(* CODESYS project WS11.project
   Title: WS11
   Version: 1.2.0
   Company: TTControl S.r.l.

Project tree, tasks and I/O mapping:
  Device : HY-TTC 580, TTControl, order no. n/a, version 1.8.0.0
    application Application
      libraries: Standard, * (System); Base Control Library Unsafe, 0.4.0.2 (TTControl); lib500_can2, 0.2.0.5 (TTControl); lib500, 1.8.0.0 (TTControl); lib500_types, 1.8.0.0 (TTControl); lib500_syscom, 1.8.0.0 (TTControl)
      task MainTask (cyclic, interval t#10ms, priority 2, watchdog t#10ms x 1) calls PLC_PRG
      task _ErrorCallback (externalevent, external event ErrorCallback, priority 1) calls _ErrorCB_PRG
      task _NotificationCallback (externalevent, external event NotificationCallback, priority 0) calls _NotificationCB_PRG
      program PLC_PRG [ST]
      program _ErrorCB_PRG [ST]
      program _NotificationCB_PRG [ST]
      global variables GVL
      program ReadMe [ST]
      program Disclaimer [ST]
      data type t_Power
      data type t_PWM
      global variables CONSTANTS
    CANs : CANs, TTControl, order no. n/a, version 1.8.0.0
      CAN0 : CAN0, TTControl, order no. n/a, version 1.8.0.0
      CAN1 : CAN1, TTControl, order no. n/a, version 1.8.0.0
          settings: Baudrate = 250
      CAN2 : CAN2, TTControl, order no. n/a, version 1.8.0.0
      CAN3 : CAN3, TTControl, order no. n/a, version 1.8.0.0
      CAN4 : CAN4, TTControl, order no. n/a, version 1.8.0.0
      CAN5 : CAN5, TTControl, order no. n/a, version 1.8.0.0
      CAN6 : CAN6, TTControl, order no. n/a, version 1.8.0.0
    System : System, TTControl, order no. n/a, version 1.8.0.0
        output Application.gPowerStage.Set.state : BYTE  // mode
        input  Application.gPowerStage.Set.error : WORD  // error
        output Application.gSafetySwitch0.Set.state : BYTE  // mode
        input  Application.gSafetySwitch0.Set.error : WORD  // error
        output Application.gSensorSupply.Set.state : BYTE  // mode
        input  Application.gSensorSupply.Set.error : WORD  // error
        input  Application.gDiagState : lib500_types.DIAG_STATUS  // diag_status
        input  Application.gSafetySwitch0.Feedback : lib500_types.IO_ADC_STATUS  // SSW0
        input  Application.gSensorSupply.Feedback : lib500_types.IO_ADC_STATUS  // SSUP0
        input  Application.gPowerStage.Get : lib500_types.IO_POWER_STATUS  // Powerstage
        input  Application.gSafetySwitch0.Get : lib500_types.IO_POWER_STATUS  // SSW0
        input  Application.gSensorSupply.Get : lib500_types.IO_POWER_STATUS  // SSUP0
        unmapped channels: mode, error, mode, error, mode, error, mode, error, shutdown, error, enable_error_group_0, enable_error_group_1, enable_error_group_2, safe_state, error, driver_init_error, UBAT, Terminal_15, WakeUp, Temperature, SSW1, SSW2, SSUP1, SSUP2, status, write, boot_error, trigger_error, SSW1, SSW2, SSUP1, SSUP2, Terminal_15, WakeUp, ExtShutOff0, ExtShutOff1, ExtShutOff2
      Analog_Inputs_2Mode_10V : AIN_2Mode_10V, TTControl, order no. n/a, version 1.8.0.0
        Pin 107
          PotRed : IoDrvADC2Mode10, TTControl, order no. n/a, version 1.8.0.0
              input  Application.gPotRed : lib500_types.IO_ADC_STATUS  // status
              unmapped channels: reset_trigger, reset_count, reset_error
        Pin 131
          <Empty>
        Pin 108
          <Empty>
        Pin 132
          <Empty>
        Pin 109
          <Empty>
        Pin 133
          <Empty>
        Pin 110
          <Empty>
        Pin 134
          <Empty>
      Analog_Inputs_2Mode_32V : AIN_2Mode_32V, TTControl, order no. n/a, version 1.8.0.0
        Pin 111
          <Empty>
        Pin 135
          <Empty>
        Pin 112
          <Empty>
        Pin 136
          <Empty>
        Pin 113
          <Empty>
        Pin 137
          <Empty>
        Pin 114
          <Empty>
        Pin 138
          <Empty>
      Analog_Inputs_3Mode : AIN_3Mode, TTControl, order no. n/a, version 1.8.0.0
        Pin 103
          <Empty>
        Pin 127
          <Empty>
        Pin 104
          <Empty>
        Pin 128
          <Empty>
        Pin 105
          <Empty>
        Pin 129
          <Empty>
        Pin 106
          <Empty>
        Pin 130
          <Empty>
      Digital_Outputs_HS : HSDOUT, TTControl, order no. n/a, version 1.8.0.0
        Pin 149
          <Empty>
        Pin 173
          <Empty>
        Pin 152
          <Empty>
        Pin 176
          <Empty>
        Pin 155
          <Empty>
        Pin 179
          <Empty>
        Pin 158
          <Empty>
        Pin 182
          <Empty>
      Digital_Outputs_LS : LSDOUT, TTControl, order no. n/a, version 1.8.0.0
        Pin 251
          <Empty>
        Pin 238
          <Empty>
        Pin 252
          <Empty>
        Pin 239
          <Empty>
        Pin 253
          <Empty>
        Pin 240
          <Empty>
        Pin 254
          <Empty>
        Pin 241
          <Empty>
      PVG_Outputs : PVG, TTControl, order no. n/a, version 1.8.0.0
        Pin 161
          <Empty>
        Pin 185
          <Empty>
        Pin 188
          <Empty>
        Pin 164
          <Empty>
        Pin 191
          <Empty>
        Pin 167
          <Empty>
        Pin 194
          <Empty>
        Pin 170
          <Empty>
      PWM_Outputs : PWM, TTControl, order no. n/a, version 1.8.0.0
        Safety_switch_0 : PWM_SSW0, TTControl, order no. n/a, version 1.8.0.0
          Pin 153
            LedRed : IoDrvPWM, TTControl, order no. n/a, version 1.8.0.0
                output Application.gLedRed.DutyCycle : WORD  // duty_cycle
                input  Application.gLedRed.Error : WORD  // error_code
                input  Application.gLedRed.PWMFeedback : lib500_types.IO_PWM_FEEDBACK  // feedback
                input  Application.gLedRed.CurrMeasurement : lib500_types.IO_PWM_CURRENT_QUEUE_E  // current
                unmapped channels: reset_trigger, reset_count, reset_error
          Pin 177
            <Empty>
          Pin 156
            <Empty>
          Pin 180
            <Empty>
          Pin 159
            <Empty>
          Pin 183
            <Empty>
          Pin 186
            <Empty>
          Pin 162
            <Empty>
          Pin 189
            <Empty>
          Pin 165
            <Empty>
          Pin 192
            <Empty>
          Pin 168
            <Empty>
          Pin 195
            <Empty>
          Pin 171
            <Empty>
        Safety_switch_1 : PWM_SSW1, TTControl, order no. n/a, version 1.8.0.0
          Pin 154
            <Empty>
          Pin 178
            <Empty>
          Pin 157
            <Empty>
          Pin 181
            <Empty>
          Pin 160
            <Empty>
          Pin 184
            <Empty>
          Pin 187
            <Empty>
          Pin 163
            <Empty>
          Pin 190
            <Empty>
          Pin 166
            <Empty>
          Pin 193
            <Empty>
          Pin 169
            <Empty>
          Pin 196
            <Empty>
          Pin 172
            <Empty>
        Safety_switch_2 : PWM_SSW2, TTControl, order no. n/a, version 1.8.0.0
          Pin 101
            <Empty>
          Pin 125
            <Empty>
          Pin 150
            <Empty>
          Pin 174
            <Empty>
          Pin 102
            <Empty>
          Pin 126
            <Empty>
          Pin 151
            <Empty>
          Pin 175
            <Empty>
      Timer_Inputs_Cur : TIN_Cur, TTControl, order no. n/a, version 1.8.0.0
        Pin 115
          <Empty>
        Pin 139
          <Empty>
        Pin 116
          <Empty>
        Pin 140
          <Empty>
        Pin 117
          <Empty>
        Pin 141
          <Empty>
      Timer_Inputs : TIN, TTControl, order no. n/a, version 1.8.0.0
        Pin 122
          <Empty>
        Pin 146
          <Empty>
        Pin 123
          <Empty>
        Pin 147
          <Empty>
        Pin 124
          <Empty>
        Pin 148
          <Empty>
*)

// Device/Application/t_Power
TYPE t_Power :
STRUCT
	// structure for POWER outputs
	Set			: lib500_types.IO_POWER_STATUS := (state := lib500_types.IO_POWER_STATE.IO_POWER_OFF);		// set power output state
	Get			: lib500_types.IO_POWER_STATUS := (state := lib500_types.IO_POWER_STATE.IO_POWER_OFF);		// get power output state 
	Feedback	: lib500_types.IO_ADC_STATUS;																// get power output voltage feetback
END_STRUCT
END_TYPE

// Device/Application/t_PWM
TYPE t_PWM :
STRUCT
	// structure for PWM outputs
	DutyCycle		: WORD := 0;								// pin duty cycle
	Error			: lib500_types.IO_ERRORTYPE;				// pin errorcode
	CurrMeasurement	: lib500_types.IO_PWM_CURRENT_QUEUE_E;		// pin current measurement
	CurrentValue	: WORD;										// usable current value
	PWMFeedback		: lib500_types.IO_PWM_FEEDBACK;				// voltage feedback
END_STRUCT
END_TYPE

// Device/Application/GVL
VAR_GLOBAL
	gDiagState 			: lib500_types.DIAG_STATUS;			// ECU diagnostic status
                                                            	
    gPowerStage     	: t_Power;							// Powerstage status structure
	gSafetySwitch0  	: t_Power;							// Safety Switch 0 status structure
    gSensorSupply       : t_Power;   						// Sensor Supply status structure
    gPotRed        		: lib500_types.IO_ADC_STATUS;       // Red Potentiometer value
    gLedRed        		: t_PWM;	                        // Led Red output
	gCan1          		: tCan;                             // Structure for sending / receiving CAN messages
END_VAR

// Device/Application/CONSTANTS
{attribute 'qualified_only'}
VAR_GLOBAL CONSTANT
	MAJOR : BYTE := 1;			// SW Version major
	MINOR : BYTE := 0;			// SW Version minor
	PATCH : BYTE := 8;			// SW Version patch
END_VAR

// Device/Application/PLC_PRG
(*****************************************************************************************
*  Copyright (C) 2022 TTControl S.r.l. All rights reserved.
*  Julius Durst Str. 66, I-39042 Brixen/Bressanone (BZ), Italy, https://ttcontrol.4me.com/
*
*  PRE: 			none
*  POST: 			none
*  GLOBAL:			gPowerStage, gSensorSupply, gSafetySwitch0, gPotRed, gLedRed, gCan1
*  LIBRARIES:		none
*  DESCRIPTION: 	This POU inizializes the powerstage and configures an analog input
*                   in voltage mode and an output in PWM mode. It reads CAN ID 0x200
*                   and set the PWM output depending on Byte 0 / 1 of this CAN message.
*                   It writes the value of analog input (Byte 0 / 1) with CAN ID 0x100. 					
*  REVISION HISTORY:	
*  2015-05-11		TLE 	Creation.
*  2016-04-05		TLE		Update to target 1.0.0.0
*  2017-02-06		TLE		Update to target 1.2.0.0
*  2017-11-27		TLE		Update to target 1.3.0.0
*  2017-04-09		ADC		Update to target 1.4.0.0
*  2019-07-23		EPI		Update to target 1.6.1.0
*  2020-11-09		EPI		Update to target 1.7.1.0
*  2022-02-21		EPI		Add diagnostic state and pin errorcodes
*  2022-07-13		EPI		Update to target 1.8.0.0
*
*****************************************************************************************)
PROGRAM PLC_PRG
VAR
	InitPLC       : BOOL := TRUE;		(* Initialization variable *)
	fbCanTxId100  : CanTx;              (* Function block to send one CAN message *)
	fbCanTxId110  : CanTx;       (* Function block to send one CAN message *)
	fbCanTxId120  : CanTx;       (* Function block to send one CAN message *)
	fbCanTxId130  : CanTx;       (* Function block to send one CAN message *)
	TxData        : ARRAY[0..7] OF BYTE;(* Data to be transmitted *)
	TxData_ID_110        : ARRAY[0..7] OF BYTE;(* Data to be transmitted *)
	TxData_ID_120_echo        : ARRAY[0..7] OF BYTE;(* Data to be transmitted *)
	TxData_ID_130_echo        : ARRAY[0..7] OF BYTE;(* Data to be transmitted *)
	fbCanRxId200  : CanRx;              (* Function block to get one CAN message*)
	
END_VAR

GVL.gDiagState.diag_state;																// update variable and display show diag state

IF (initPLC = TRUE) THEN
	GVL.gPowerStage.Set.state    	:= lib500_types.IO_POWER_STATE.IO_POWER_ON;	    	// Switching on Power Stage
    GVL.gSafetySwitch0.Set.state 	:= lib500_types.IO_POWER_STATE.IO_POWER_ON;      	// Switching on Safety Switch for PWM use
	GVL.gSensorSupply.Set.state 	:= lib500_types.IO_POWER_STATE.IO_POWER_ON;       	// Switching on Sensor Supply
// use variables and show values
	// Power outputs
	GVL.gPowerStage.Set.error;															// Power Stage set error
	GVL.gPowerStage.Get.state;															// Power Stage get state
	GVL.gPowerStage.Feedback.value;														// Power Stage voltage feedback
	GVL.gSafetySwitch0.Set.error;														// Safety Switch set error
	GVL.gSafetySwitch0.Get.state;														// Safety Switch get state
	GVL.gSafetySwitch0.Feedback.value;													// Safety Switch voltage feedback
	GVL.gSensorSupply.Set.error;														// Sensor Supply set error
	GVL.gSensorSupply.Get.state;														// Sensor Supply get state
	GVL.gSensorSupply.Feedback.value;													// Sensor Supply voltage feedback
	// application IOs
	GVL.gPotRed.error;																	// Pot Red pin error
	GVL.gLedRed.Error;																	// Led Red pin error
	GVL.gLedRed.CurrMeasurement.error;													// Led Red current measurement error
	GVL.gLedRed.CurrMeasurement.values[0];												// Led Red current
	GVL.gLedRed.PWMFeedback.high_time;													// Led Red PWM feedback
	
// Initialize CAN 1	
	CanInit(	iEnable			:= TRUE,                                				// Initialiaze CAN 
				iChannel		:= 1, 													// CAN Channel 1
				iCAN			:= ADR(GVL.gCan1), 										// Structure for sending / receiving CAN messages
				iBaudrate       := 500, 												// 250 kBit
				iCanIdExtended  := FALSE, 												// Standard CAN Frame
				iEcuCycleTime   := T#10MS);												// Cycle time of task calling TX and RX
    InitPLC := FALSE;																	// Execute this block one time for initialisation
END_IF                                                                  				
                                                                        				
cl_split_word(	input	:= DWORD_TO_WORD(GVL.gPotRed.value),							// Split PotRed value in two bytes to send them over CAN
				byte0	=> TxData[0],                                   				
				byte1	=> TxData[1]);                                  				
				                                                        				
fbCanTxId100(	iEnable				:= TRUE, 											// Enables sending of messages
				iCAN				:= ADR(GVL.gCan1),									// Structure for sending / receiving CAN messages
				iForceSend			:= FALSE,                           				// Force sending sends message immediately
				iTransmitRate		:= T#100MS, 										// Cyclic transmission every 100ms
				iCanId				:= 16#100,											// CAN Id for message to send
				iCanIdExtended		:= FALSE, 											// Standard CAN Frame
				iByteCount			:= 8,												// Number of bytes to send
				iData				:= TxData, 											// Data frame
				oTransmitterId		=> ,                                				
				oTooManyTransmitters=> ,                                				
				oMsgSent			=> );        
				
				TxData_ID_110[0] := 15;
				TxData_ID_110[1] := 14;
				TxData_ID_110[2] := 13;
				TxData_ID_110[3] := 12;
				TxData_ID_110[4] := 11;
				TxData_ID_110[5] := 10;
				TxData_ID_110[6] := 9;
				TxData_ID_110[7] := 8;
				
fbCanTxId110(	iEnable				:= TRUE, 											// Enables sending of messages
				iCAN				:= ADR(GVL.gCan1),									// Structure for sending / receiving CAN messages
				iForceSend			:= FALSE,                           				// Force sending sends message immediately
				iTransmitRate		:= T#100MS, 										// Cyclic transmission every 100ms
				iCanId				:= 16#110,											// CAN Id for message to send
				iCanIdExtended		:= FALSE, 											// Standard CAN Frame
				iByteCount			:= 8,												// Number of bytes to send
				iData				:= TxData_ID_110, 									// Data frame
				oTransmitterId		=> ,                                				
				oTooManyTransmitters=> ,                                				
				oMsgSent			=> );                 

fbCanTxId120(	iEnable				:= TRUE, 											// Enables sending of messages
				iCAN				:= ADR(GVL.gCan1),									// Structure for sending / receiving CAN messages
				iForceSend			:= FALSE,                           				// Force sending sends message immediately
				iTransmitRate		:= T#100MS, 										// Cyclic transmission every 100ms
				iCanId				:= 16#130,											// CAN Id for message to send
				iCanIdExtended		:= FALSE, 											// Standard CAN Frame
				iByteCount			:= 8,												// Number of bytes to send
				iData				:= TxData_ID_130_echo, 									// Data frame
				oTransmitterId		=> ,                                				
				oTooManyTransmitters=> ,                                				
				oMsgSent			=> );                  
                         				        				
				                                                        				
fbCanRxId200(	iCAN				:= ADR(GVL.gCan1),  								// Structure for sending / receiving CAN messages
				iCanId				:= 16#200,											// CAN Id of receiving message 
				iCanIdExtended		:= FALSE,  											// Standard CAN Frame
				iTimeoutLimit		:= T#500MS,											// Timeout after 500ms - Flag will be set 
				oByteCount			=> ,                                	
				oData				=> ,                                	
				oNewData			=> ,                                	
				oCanTimeout			=> ,                                	
				oReceiverId			=> ,                                	
				oTooManyReceivers	=> );	                            	
                                                                        	
IF fbCanRxId200.oNewData THEN															// If new CAN data is available
	GVL.gLedRed.DutyCycle := cl_make_word(	byte0 := fbCanRxId200.oData[0], 			// Make word using two over CAN received bytes and set it as LedRed setpoint*)
											byte1 := fbCanRxId200.oData[1]);					
	
	
ELSIF fbCanRxId200.oCanTimeout THEN														// If timeout flag is enabled switch off LedRed
	GVL.gLedRed.DutyCycle := 0;
END_IF

END_PROGRAM

// Device/Application/_ErrorCB_PRG
PROGRAM _ErrorCB_PRG
VAR
	diag_state : lib500_types.DIAG_STATETYPE := lib500_types.DIAG_STATETYPE.DIAG_STATE_DISABLED;
	watchdog_state : lib500_types.DIAG_WD_STATETYPE := lib500_types.DIAG_WD_STATETYPE.DIAG_WD_STATE_UNKNOWN;
	error : lib500_types.DIAG_ERRORCODE := (error_code := lib500_types.DIAG_ERRORTYPE.DIAG_E_NOERROR, 
                                            device_num := lib500_types.DIAG_DEVICETYPE.DIAG_DEV_NONE,
                                            faulty_value := 0);
	return_code : lib500_types.IO_ERRORTYPE := lib500_types.IO_ERRORTYPE.IO_E_UNKNOWN;
	
	reaction : lib500_types.DIAG_REACTION := lib500_types.DIAG_REACTION.DIAG_ERR_SAFESTATE;
	
	call_count : UDINT := 0;
END_VAR

(* get the reason for the error callback *)
return_code := lib500.DIAG_CDS_GetErrorReason(ADR(diag_state), 
                                              ADR(watchdog_state),
                                              ADR(error));

(* custom handler code can be placed here *)

(* the choices for the reactions are:
   -> lib500_types.DIAG_REACTION.DIAG_ERR_NOACTION
   -> lib500_types.DIAG_REACTION.DIAG_ERR_SAFESTATE
   -> lib500_types.DIAG_REACTION.DIAG_ERR_DISABLE_SSW0
   -> lib500_types.DIAG_REACTION.DIAG_ERR_DISABLE_SSW1
   -> lib500_types.DIAG_REACTION.DIAG_ERR_DISABLE_SSW2
   -> lib500_types.DIAG_REACTION.DIAG_ERR_DISABLE_HS00
   -> lib500_types.DIAG_REACTION.DIAG_ERR_DISABLE_HS01
   -> lib500_types.DIAG_REACTION.DIAG_ERR_DISABLE_HS02
   -> lib500_types.DIAG_REACTION.DIAG_ERR_DISABLE_HS03
   -> lib500_types.DIAG_REACTION.DIAG_ERR_DISABLE_HS04
   -> lib500_types.DIAG_REACTION.DIAG_ERR_DISABLE_HS05
   -> lib500_types.DIAG_REACTION.DIAG_ERR_DISABLE_HS06
   -> lib500_types.DIAG_REACTION.DIAG_ERR_DISABLE_HS07
   
   it's also possible to combine (binary-or) reactions, like:
   -> lib500_types.DIAG_REACTION.DIAG_ERR_DISABLE_SSW0 OR 
      lib500_types.DIAG_REACTION.DIAG_ERR_DISABLE_SSW1
*)

(* pass the error reaction to the DIAG system *)
lib500.DIAG_CDS_SetErrorReaction(reaction);

(* increment call count *)
call_count := call_count + 1;

END_PROGRAM

// Device/Application/_NotificationCB_PRG
PROGRAM _NotificationCB_PRG
VAR
	diag_state : lib500_types.DIAG_STATETYPE := lib500_types.DIAG_STATETYPE.DIAG_STATE_DISABLED;
	watchdog_state : lib500_types.DIAG_WD_STATETYPE := lib500_types.DIAG_WD_STATETYPE.DIAG_WD_STATE_UNKNOWN;
	error : lib500_types.DIAG_ERRORCODE := (error_code := lib500_types.DIAG_ERRORTYPE.DIAG_E_NOERROR, 
                                            device_num := lib500_types.DIAG_DEVICETYPE.DIAG_DEV_NONE,
                                            faulty_value := 0);
	return_code : lib500_types.IO_ERRORTYPE := lib500_types.IO_ERRORTYPE.IO_E_UNKNOWN;
	
	call_count : UDINT := 0;
END_VAR

(* get the reason for the notification callback *)
return_code := lib500.DIAG_CDS_GetNotificationReason(ADR(diag_state), 
                                                     ADR(watchdog_state),
                                                     ADR(error));

(* custom handler code can be placed here *)

(* increment call count *)
call_count := call_count + 1;

END_PROGRAM

// Device/Application/ReadMe
(*****************************************************************************************
*  Copyright (C) 2022 TTControl S.r.l. All rights reserved.
*  Julius Durst Str. 66, I-39042 Brixen/Bressanone (BZ), Italy, https://ttcontrol.4me.com/
*
*  PRE: 			none
*  POST: 			none
*  GLOBAL:			none
*  LIBRARIES:		none
*  DESCRIPTION: 	This POU describes the use of this workshop example.
*					
*  REVISION HISTORY:	
*  2015-05-11		TLE 	Creation.
*  2016-04-05		TLE		Update to target 1.0.0.0
*  2017-02-06		TLE		Update to target 1.2.0.0
*  2017-11-27		TLE		Update to target 1.3.0.0
*  2017-04-09		ADC		Update to target 1.4.0.0
*  2019-07-23		EPI		Update to target 1.6.1.0
*  2020-11-09		EPI		Update to target 1.7.1.0
*  2022-02-21		EPI		Add diagnostic state and pin errorcodes
*  2022-07-13		EPI		Update to target 1.8.0.0
*
*****************************************************************************************)
PROGRAM ReadMe

(* * * * * * * * * * * * * * * * * * * * * * * * * * * * * * * * * * * * * * * * * * 
 *	READ ME			READ ME			READ ME			READ ME			READ ME               
 * * * * * * * * * * * * * * * * * * * * * * * * * * * * * * * * * * * * * * * * * * 
 * 
 *  This program shows how to read and write CAN 2.0b messages. It uses Pin 103
 *  as voltage mode input and Pin 153 as PWM output.
 *	
 * * * * * * * * * * * * * * * * * * * * * * * * * * * * * * * * * * * * * * * * * * )

END_PROGRAM

// Device/Application/Disclaimer
(*****************************************************************************************
*  Copyright (C) 2022 TTControl S.r.l. All rights reserved.
*  Julius Durst Str. 66, I-39042 Brixen/Bressanone (BZ), Italy, https://ttcontrol.4me.com/
*
*  PRE: 			none
*  POST: 			none
*  GLOBAL:			none
*  LIBRARIES:		none
*  DESCRIPTION: 	Disclaimer
*					
*  REVISION HISTORY:	
*  2017-01-31		TLE 	Creation.
*
*****************************************************************************************)

PROGRAM Disclaimer
VAR
END_VAR

(* * * * * * * * * * * * * * * * * * * * * * * * * * * * * * * * * * * * * * * * * * 
 *	DISCLAIMER		DISCLAIMER		DISCLAIMER		DISCLAIMER  	DISCLAIMER       
 * * * * * * * * * * * * * * * * * * * * * * * * * * * * * * * * * * * * * * * * * *  
 
This document is proprietary to TTControl GmbH and no ownership rights are hereby transferred.
No part of this document shall be used, reproduced, translated, converted, adapted, stored in an
information storage or a retrieval system, communicated or transmitted in any form or by any means
(electronic or mechanical, including photocopying, recording), for any commercial purpose, including
without limitation, sale, resale, license, rental or lease, without the prior express written consent
of TTControl GmbH.

TTControl GmbH does not make any representations, warranties or guarantees, express or implied,
as to the accuracy or completeness of the document. The information in this document is subject to
change without notice and does not represent a commitment on the part of TTControl GmbH. Users
must be aware that updates and amendments will be made from time to time to the document. It is
the user’s responsibility to determine whether there have been any such updates or amendments.
Neither TTControl GmbH nor any of its directors, officers, employees or agents shall be liable in
contract, tort or in any other manner whatsoever to any person for any loss, damage, injury, liability,
cost or expense of any nature, including without limitation incidental, special, direct or consequential
damages arising out of or in connection with the use of this document.


Der Inhalt dieses Dokuments ist geistiges Eigentum der TTControl GmbH und es werden hieran keine Eigentumsrechte 
übertragen. Dieses Dokument, einschließlich seiner Teile, darf in keiner Form und auf keine Weise (elektronisch 
oder mechanisch, einschließlich Fotokopien und Aufnahmen) füR kommerzielle Zwecke  verwendet, vervielfältigt, 
übersetzt, verändert oder adaptiert werden. "Kommerzielle Zwecke" umfassen insbesondere Verkauf, Weiterverkauf, 
Lizenz, Miete oder Pacht ohne die vorherige ausdrückliche schriftliche Zustimmung von TTControl GmbH. Es ist nicht 
erlaubt dieses Dokument, einschließlich seiner Teile, in einem Datenspeicher oder einem Datenabfragesystem zu 
speichern, es zu übertragen oder zu versenden. 

TTControl GmbH übernimmt, soweit gesetzlich zulässig, weder ausdrücklich noch stillschweigend Gewährleistungen 
oder Garantien betreffend die Richtigkeit oder Vollständigkeit des Dokuments. Die TTControl behäLT sich das Recht 
vor, ohne Benachrichtigung den Inhalt des Dokuments abzuändern, ohne dass ihr hieraus irgendwelche Verpflichtungen 
erwachsen. Der Benutzer muss sich bewusst sein, dass Aktualisierungen und Anpassungen gelegentlich erfolgen werden. 
Es obliegt dem Benutzer festzustellen, ob solche Aktualisierungen oder Anpassungen erfolgt sind. Soweit gesetzlich 
zulässig, haftet weder die TTControl GmbH noch einer ihrer Geschäftsführer, Angestellten  oder Repräsentanten vertraglich, 
schadenersatzrechtlich oder auf irgendeiner anderen Grundlage füR Verluste, Schäden,  Kosten oder Ausgaben jeglicher Art, 
einschließlich, aber nicht beschränkt auf Neben-, Folge- oder Sonderschäden, direkte oder indirekte Schäden, die aus oder 
im Zusammenhang mit diesem Dokument entstehen.

 * * * * * * * * * * * * * * * * * * * * * * * * * * * * * * * * * * * * * * * * * * 
 *	DISCLAIMER		DISCLAIMER		DISCLAIMER		DISCLAIMER  	DISCLAIMER               
 * * * * * * * * * * * * * * * * * * * * * * * * * * * * * * * * * * * * * * * * * *)

END_PROGRAM
